{attribute 'qualified_only'}
{attribute 'strict'}
{attribute 'to_string'}
TYPE E_ModuleState :
(
    IDLE,
    SET_DIRECTION,
    MOVE_PART,
    WAIT_FOR_MEASUREMENT,
    EXECUTING_MEASUREMENT,
    WAIT_FOR_FOLLOWER,
    TRANSFER_TO_FOLLOWER,
    CLEAR_CONVEYOR,
    LOCKOUT
);
END_TYPE

(* stored: Version 1.1.0.1
   DUT E_ModuleState: Id {9fa85e8d-2ad3-4648-afbb-d5b75f43373c} *)
